FUNCTION TryConvert_ULINT_TO_INT : BOOL
VAR_INPUT
	in : ULINT;
	out : REFERENCE TO INT;
END_VAR

IF in > DatatypeLimits.MAX_VALUE_OF_ULINT_WHICH_CAN_BE_HELD_IN_A_INT THEN
	RETURN;
END_IF

out := ULINT_TO_INT(in);
TryConvert_ULINT_TO_INT := TRUE;

END_FUNCTION

(* stored: Version 1.1.0.1, ProductVersion 3.1.4024.12
   POU TryConvert_ULINT_TO_INT: Id {3bce4815-0b00-42f7-9b5a-433a3d997a39}, SpecialFunc None *)
